// TIA Portal V17 export
// export: Created 2025-06-26T06:49:18.1843279Z, ExportSetting WithDefaults, DisplayName Totally Integrated Automation Portal, DisplayVersion V17 Update 8, DisplayName TIA Portal Openness, DisplayVersion V17 Update 8, DisplayName TIA Portal Version Control Interface, DisplayVersion V17, DisplayName STEP 7 Professional, DisplayVersion V17 Update 8, DisplayName STEP 7 Safety, DisplayVersion V17 Update 6, DisplayName WinCC Advanced, DisplayVersion V17 Update 8
FUNCTION "States" : Void   // FC27, FBD
TITLE = State change signal generation
{ S7_Optimized_Access := 'TRUE' }
VERSION : 0.1
// stored: AutoNumber true, IsIECCheckEnabled false, SetENOAutomatically false, UDAEnableTagReadback false
BEGIN

REGION Network 1: State 0 Initialization
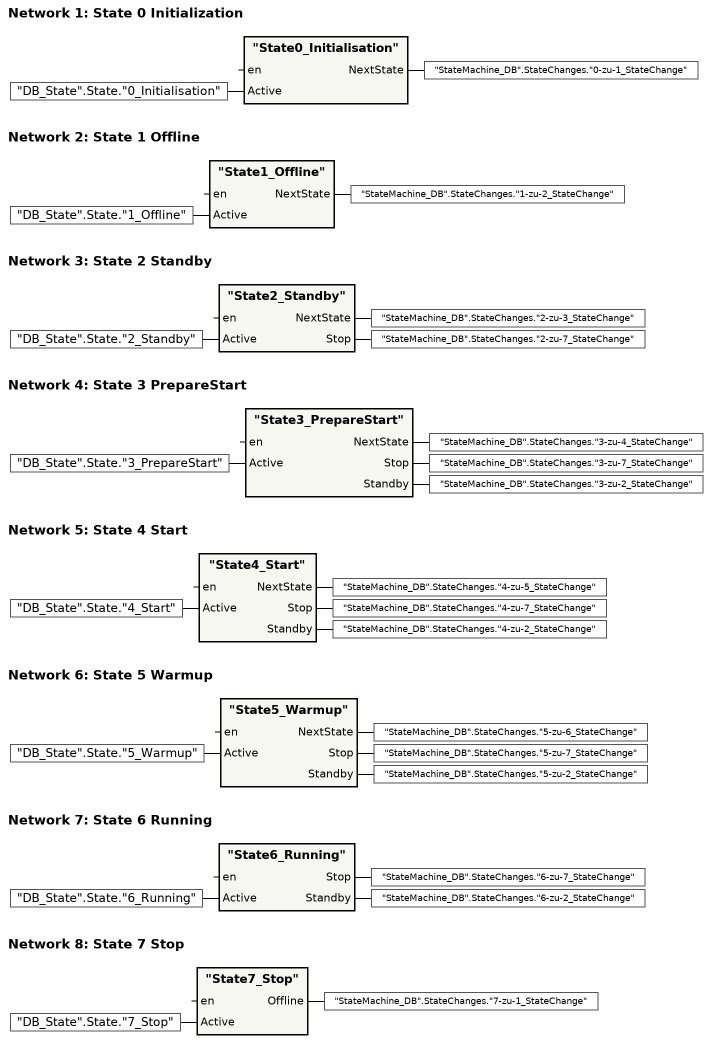
   "State0_Initialisation"(Active := "DB_State".State."0_Initialisation",
                           NextState => "StateMachine_DB".StateChanges."0-zu-1_StateChange");
END_REGION

REGION Network 2: State 1 Offline
   "State1_Offline"(Active := "DB_State".State."1_Offline",
                    NextState => "StateMachine_DB".StateChanges."1-zu-2_StateChange");
END_REGION

REGION Network 3: State 2 Standby
   "State2_Standby"(Active := "DB_State".State."2_Standby",
                    NextState => "StateMachine_DB".StateChanges."2-zu-3_StateChange",
                    Stop => "StateMachine_DB".StateChanges."2-zu-7_StateChange");
END_REGION

REGION Network 4: State 3 PrepareStart
   "State3_PrepareStart"(Active := "DB_State".State."3_PrepareStart",
                         NextState => "StateMachine_DB".StateChanges."3-zu-4_StateChange",
                         Stop => "StateMachine_DB".StateChanges."3-zu-7_StateChange",
                         Standby => "StateMachine_DB".StateChanges."3-zu-2_StateChange");
END_REGION

REGION Network 5: State 4 Start
   "State4_Start"(Active := "DB_State".State."4_Start",
                  NextState => "StateMachine_DB".StateChanges."4-zu-5_StateChange",
                  Stop => "StateMachine_DB".StateChanges."4-zu-7_StateChange",
                  Standby => "StateMachine_DB".StateChanges."4-zu-2_StateChange");
END_REGION

REGION Network 6: State 5 Warmup
   "State5_Warmup"(Active := "DB_State".State."5_Warmup",
                   NextState => "StateMachine_DB".StateChanges."5-zu-6_StateChange",
                   Stop => "StateMachine_DB".StateChanges."5-zu-7_StateChange",
                   Standby => "StateMachine_DB".StateChanges."5-zu-2_StateChange");
END_REGION

REGION Network 7: State 6 Running
   "State6_Running"(Active := "DB_State".State."6_Running",
                    Stop => "StateMachine_DB".StateChanges."6-zu-7_StateChange",
                    Standby => "StateMachine_DB".StateChanges."6-zu-2_StateChange");
END_REGION

REGION Network 8: State 7 Stop
   "State7_Stop"(Active := "DB_State".State."7_Stop",
                 Offline => "StateMachine_DB".StateChanges."7-zu-1_StateChange");
END_REGION
END_FUNCTION
